// TIA Portal project "project_counter_application_sim" (V16)

(* hardware
DEVICE "S7-1200 station_1"  S7-1200 Station
   slot 0: "Rack_0"  S7-1200 Rack  Rack  V1.0
   slot 1: "PLC_1"  CPU 1214C DC/DC/Rly  6ES7 214-1HG40-0XB0  V4.4
*)

// ===== PLC "PLC_1"  CPU 1214C DC/DC/Rly =====

VAR_GLOBAL   // PLC tag table "Default tag table"
   ""START BUT"" AT %I0.0 : Bool;
   ""TERMİK 1"" AT %I0.2 : Bool;
   ""TERMİK 2"" AT %I0.3 : Bool;
   ""TERMİK 3"" AT %I0.4 : Bool;
   ""MOTOR-2"" AT %Q0.1 : Bool;
   ""MOTOR-3"" AT %Q0.2 : Bool;
   ""MOTOR-1"" AT %Q0.0 : Bool;
END_VAR